PROGRAM MAIN
VAR
	fb_pmlstatemachine_Testsuite : FB_PMLStateMachine_Tests;
END_VAR

TcUnit.RUN_IN_SEQUENCE();

END_PROGRAM

(* stored: Version 1.1.0.1, ProductVersion 3.1.4024.11
   POU MAIN: Id {3619bd3f-fc5b-432b-85a8-108cc19a861e}, SpecialFunc None *)
